INTERFACE I_HostExtensions EXTENDS __SYSTEM.IQueryInterface

PROPERTY Extensions : I_Extensions
GET
END_GET
END_PROPERTY

END_INTERFACE

(* stored: Version 1.1.0.1, ProductVersion 3.1.4024.12
   Itf I_HostExtensions: Id {2c4d3330-a4d5-0bf1-1982-102b528ecb24}
   Property Extensions: Id {a2b464af-5b46-4255-b253-1cd7aa283d6e}
   Get Get: Id {5621afa0-ca92-4e9c-9f98-7a2cc6188420} *)
